//Robot:
//This FB represents the robot and links the control algorithm with the physical I/O of the robot. It is implemented in a separate FB so it is easily interchangeable with
//simulated robot whenever needed. 
FUNCTION_BLOCK Robot
VAR_INPUT
	enable: BOOL;
	vXref, vYref, vThetaRef: LREAL;
END_VAR
VAR_OUTPUT
	vX, vY, vTheta: LREAL;
	sliderGotTriggered: BOOL;
	bumperGotTriggered: BOOL;
END_VAR
VAR
	sliderTrigger: F_TRIG;
	bumperTrigger: R_TRIG;
	//inputs to robot
	vXtoRobot 		AT%Q*: LREAL;
	vYtoRobot		AT%Q*: LREAL;
	vThetaToRobot 	AT%Q*: LREAL;
	
	//outputs from robot
	slider 			AT%I*: BOOL;
	bumper			AT%I*: BOOL;
	vel: 	VelocityMeasurement;
	i1_raw, i2_raw, i3_raw	AT%I*: 					UINT;
	i1, i2, i3 : INT;
END_VAR

vel();

sliderTrigger(CLK := slider, Q => sliderGotTriggered);
bumperTrigger(CLK := bumper, Q => bumperGotTriggered);

vX 		:= vel.vXRobot;
vY 		:= vel.vYRobot;
vTheta  := vel.vThetaRobot;

//write control outputs to robot if enabled
IF enable = TRUE THEN
			vXtoRobot     := vXref;
			vYtoRobot	  := vYref;
			vThetaToRobot := vThetaRef;
ELSE
			vXtoRobot     := 0;
			vYtoRobot	  := 0;
			vThetaToRobot := 0;
END_IF

i1 := UINT_TO_INT(i1_raw);
i2 := UINT_TO_INT(i2_raw);
i3 := UINT_TO_INT(i3_raw);

END_FUNCTION_BLOCK

(* stored: Version 1.1.0.1, ProductVersion 3.1.4024.11
   POU Robot: Id {c2c95814-6e9d-4a67-9cd4-cf68c7267fb5}, SpecialFunc None *)
